{attribute 'qualified_only'}
{attribute 'strict'}
TYPE stGRID_POS :
(
	poi := 0,
	pu := 1
);
END_TYPE

(* stored: Version 1.1.0.1, ProductVersion 3.1.4026.11
   DUT stGRID_POS: Id {c0750ff1-87a1-43cc-ae44-2081110f86f5} *)
